// TIA Portal project "Zufallszahl" (V20)

(* hardware
DEVICE "S7-1500/ET200MP-Station_1"  S7-1500 station
   slot 0: "Profilschiene_0"  Rack  6ES7 590-1***0-0AA0
   slot 1: "PLC_1"  CPU 1513-1 PN  6ES7 513-1AM03-0AB0  V4.0
      slot 3: "CPU-Display_1"  6ES7591-1AA00-0AA0
      slot 32768: "PROFINET-Schnittstelle_1"  X1
         slot 32769: "Port_1"  X1 P1
         slot 32770: "Port_2"  X1 P2
      slot 34817: "Virtual CP interface port_1"  Virtual CP interface port  Virtual CP interface port FW V4.0
   slot 2: "DI 16x24VDC BA_1"  DI 16x24VDC BA  6ES7 521-1BH10-0AA0  V1.1
   slot 3: "DQ 16x24VDC/0.5A ST_1"  DQ 16x24VDC/0.5A ST  6ES7 522-1BH00-0AB0  V2.0
   slot 4: "AI 8xU/I/R/RTD BA_2"  AI 8xU/I/R/RTD BA  6ES7 531-7QF00-0AB0  V1.0
   slot 5: "AQ 8xU/I HS_2"  AQ 8xU/I HS  6ES7 532-5HF00-0AB0  V2.2
*)

// ===== PLC "PLC_1"  CPU 1513-1 PN =====

DATA_BLOCK "Zufallszahl_DB"   // DB1
{ S7_Optimized_Access := 'TRUE' }
VERSION : 0.1
// stored: InstanceOfName Zufallszahl
"Zufallszahl"
BEGIN
END_DATA_BLOCK

FUNCTION_BLOCK "Zufallszahl"   // FB1, FBD
{ S7_Optimized_Access := 'TRUE' }
VERSION : 0.1
   VAR
      Zufallszahl_Generator : Struct
         Zufallszahl : DInt;
         Fehler : Struct
            Aktiv : Bool;
            Status : Word;
            UnterfunkionStatus : Word;
         END_STRUCT;
      END_STRUCT;
   END_VAR
   VAR CONSTANT
      Untere_Grenze : DInt := 100;
      Obere_Grenze : DInt := 999;
   END_VAR
BEGIN

REGION Network 1
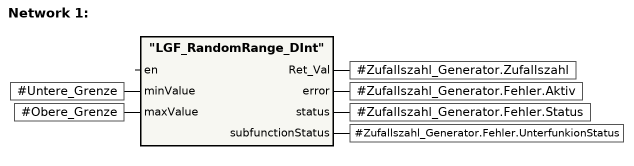
   #Zufallszahl_Generator.Zufallszahl := "LGF_RandomRange_DInt"(minValue := #Untere_Grenze,
                           maxValue := #Obere_Grenze,
                           error => #Zufallszahl_Generator.Fehler.Aktiv,
                           status => #Zufallszahl_Generator.Fehler.Status,
                           subfunctionStatus => #Zufallszahl_Generator.Fehler.UnterfunkionStatus);
END_REGION
END_FUNCTION_BLOCK

ORGANIZATION_BLOCK "Main"   // OB1, FBD, ProgramCycle
TITLE = "Main Program Sweep (Cycle)"
{ S7_Optimized_Access := 'TRUE' }
VERSION : 0.1
   VAR_INPUT
      Initial_Call : Bool;   // Initial call of this OB
      Remanence : Bool;   // =True, if remanent data are available
   END_VAR
   VAR_TEMP
      Aktuelle_Zeit : DTL;
      Fehler : Word;
   END_VAR
BEGIN

REGION Network 1
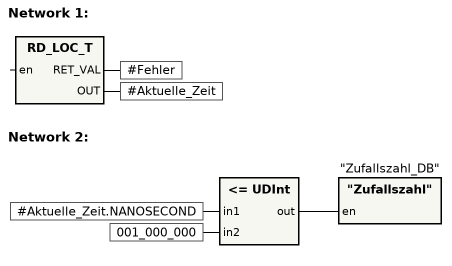
   #Fehler := RD_LOC_T(OUT => #Aktuelle_Zeit);
END_REGION

REGION Network 2
   IF #Aktuelle_Zeit.NANOSECOND <= 001_000_000 THEN
       "Zufallszahl_DB"();   // "Zufallszahl"
   END_IF;
END_REGION
END_ORGANIZATION_BLOCK

// folder: LGF/04 Math operations

FUNCTION "LGF_RandomRange_DInt" : DInt   // FC10013, SCL
TITLE = LGF_RandomRange_DInt
{ S7_Optimized_Access := 'TRUE' }
AUTHOR : Siemens_Digital_Industries
FAMILY : LGF
NAME : LGF_RandomRange_DInt
// This function generates a random value in defined limits with each call.  
// The random number has the data type DInt in the specified range.
// Diese Funktion generiert bei jedem Aufruf einen zufälligen Wert zwischen einem definierten Max- und Minwert.  
// Die Zufallszahl hat den Datentyp DInt im spezifiziertem Wertebereich.
   VAR_INPUT
      minValue : DInt;   // Minimalwert der für den Wertebereich der Zufallszahl - Untergrenze / Minimum value of the range of the random number - lower border
      maxValue : DInt;   // Maximalwert der für den Wertebereich der Zufallszahl - Obergrenze / Maximum value of the range of the random number - upper border
   END_VAR
   VAR_OUTPUT
      error : Bool;   // FALSE: No error TRUE: An error occurred during the execution of the FB / FALSE: Kein Fehler TRUE: Während der Ausführung des FB ist ein Fehler aufgetreten
      status : Word;   // 16#0000-16#7FFF: Status of the FB 16#8000-16#FFFF: Error identification (see following Table) / 16#0000-16#7FFF: Status des FB 16#8000-16#FFFF: Fehleridentifikation (siehe folgende Tabelle)
      subfunctionStatus : Word;   // Status or return value of called FB's, FC's and system blocks / Status oder Rückgabewert von aufgerufenen FB's / FC's und Systemfunktionen
   END_VAR
   VAR_TEMP
      tempTime : DTL;   // Temp memory for System time / Temp variable für System Zeit
      tempNanoSecondInDWord : DWord;   // Temp UDInt converted to DWord for access to individual bytes / Temp UDInt konvertiert nach Dword für den Zufriff per Slice auf die Bytes
      tempTimeStatus : Word;   // Temp status of the instruction `RD_SYS_T` / Temp Status der Systemfunktion `RD_SYS_T`
      tempRandomValue : DWord;   // Temp Random startvalue / Temp Zufallswert als Startwert
      tempNormReal : Real;   // Temp normalized Real value (0.0 - 1.0) / Temp Normalisierer Realwert (0.0 - 1.0)
   END_VAR
   // Ret_Val : Random Real number in the predefined range / Zufallszahl vom Datentyp Real im definierten Wertebereich
   VAR CONSTANT
      ZERO : DInt := 0;   // Zero / 0.0 - value in case of error / Null / 0.0 - Rückgabewert im Fehlerfall
      MAX_UDINT : UDInt := 4294967295 ;   // Maximum DInt datatype / Maximalwert eines DInt Datentype
      SUB_STATUS_NO_ERROR : Word := 16#0000;   // Status: sub function call ends without error / Status: Unterfunktionsaufruf ohne Fehler beendet
      STATUS_FINISHED_NO_ERROR : Word := 16#0000;   // Execution finished without errors / Abarbeitung ohne Fehler beendet
      ERR_MAX_LESS_MIN : Word := 16#8200;   // Error: The ranges specified are wrong: `minValue` is greater than `maxValue` / Fehler: Der spezifizierte Wetebereich is fehlerhaft: `minValue` ist größer als `maxValue`
      ERR_RD_SYS_T : Word := 16#8600;   // Error in `RD_SYS_T` command - check `subFunctionStatus` code / Fehler in Anweisung `RD_SYS_T` - weitere infos in `subFunctionStatus`
   END_VAR
BEGIN
   REGION Block info header
     //=============================================================================
     // SIEMENS AG / (c)Copyright 2017
     //-----------------------------------------------------------------------------
     // Title:            LGF_RandomRange_DInt
     // Comment/Function: This function generates random numbers in defined limits (Datatype DInt)
     // Library/Family:   LGF(Library General Functions)
     // Author:           Siemens Digital Industry Support
     // Tested with:      S7-PLCSIM Advanced V2.0 SP1
     // Engineering:      TIA Portal V15 Update 2
     // Restrictions:     ENO disabled - error handling done by error and status
     // Requirements:     PLC (S7-1200 / S7-1500)
     //-------------------------------------------------------------------------------
     // Change log table:
     // Version  | Date       | Expert in charge       | Changes applied
     //----------|------------|------------------------|------------------------------
     // 01.00.00 19.08.2015  Siemens Industry Online Support
     //                      First released version
     // 01.00.01 02.01.2017  Siemens Industry Online Support
     //                      Upgrade: TIA Portal V14 Update 1
     // 01.00.02 17.08.2018  Siemens Industry Online Support
     //                      Upgrade: TIA V15 Update 2
     // 01.00.03 23.11.2018  Siemens Industry Online Support
     //                      Upgrade: TIA V15.1
     // 01.01.00 09.10.2019  Simatic Systems Support
     //                      Renamed from "LGF_RandomInt" to "LGF_RandomRange_DInt"
     //                      change random datatype from Int to DInt
     //                      Regions, comments and constants are added
     // 03.00.00 23.04.2020  Simatic Systems Support
     //                      Set version to V3.0.0, harmonize the version of the whole library
     // 03.00.01 04.02.2021  Simatic Systems Support
     //                      Insert documentation
     //=============================================================================
   END_REGION Block info header

   REGION DESCRIPTION
     (/*Note
   :    The status of called commands is output in `subFunctionStatus`. In this case, the output value in `status` indicates which command caused the error. In this case, refer to the TIA Portal Online Help section for information on the respective commands.

   The block generates random values that are between the specified `minValue` and the `maxValue`. This random value is output via the `Ret_Val`.

   The random value is formed from the nanoseconds of the current system time of the CPU. The byte order of this value is inverted and then converted to a DInt.
   Hinweis
   :    In `subFunctionStatus` wird der Status von aufgerufenen Anweisungen ausgegeben. Der Ausgangswert in `status` gibt in diesem Fall an, welche Anweisung den Fehler verursacht hat. Holen Sie sich in diesem Fall die Informationen aus der TIA Portal Online Hilfe zu den jeweiligen Anweisungen.

   Der Baustein generiert zufällige Werte, die zwischen dem angegebenen `minValue`-Wert und `maxValue`-Wert liegen. Dieser zufällige Wert wird über den `Ret_Val` ausgegeben.

   Der Zufallswert wird aus den Nanosekunden der aktuellen Systemzeit der CPU gebildet. Dabei wird die Bytereihenfolge dieses Wertes invertiert und anschließend in eine DInt ungewandelt.*/)
   END_REGION DESCRIPTION

   REGION Validation
     // Check if the maximal Value is less than the minimal value
     IF (#minValue > #maxValue) THEN
       #error := true;
       #status := #ERR_MAX_LESS_MIN;
       #subfunctionStatus := #SUB_STATUS_NO_ERROR;
       #LGF_RandomRange_DInt := #ZERO;
       RETURN;
     END_IF;

     // Read system time
     #tempTimeStatus := INT_TO_WORD(RD_SYS_T(#tempTime));

     // Check return variable for error
     IF (#tempTimeStatus <> #SUB_STATUS_NO_ERROR) THEN
       #error := true;
       #status := #ERR_RD_SYS_T;
       #subfunctionStatus := #tempTimeStatus;
       #LGF_RandomRange_DInt := #ZERO;
       RETURN;
     END_IF;
   END_REGION

   REGION Calculating random number
     // Converting to double word so individual bytes can be addressed
     #tempNanoSecondInDWord := UDINT_TO_DWORD(#tempTime.NANOSECOND);

     // Callculate a random-start-value depending on the time
     #tempRandomValue.%B3 := #tempNanoSecondInDWord.%B0;
     #tempRandomValue.%B2 := #tempNanoSecondInDWord.%B1;
     #tempRandomValue.%B1 := #tempNanoSecondInDWord.%B2;
     #tempRandomValue.%B0 := #tempNanoSecondInDWord.%B3;

     // Norm the calculated random number: 0.0 <= #tempNormReal <= 1.0
     #tempNormReal := UDINT_TO_REAL(DWORD_TO_UDINT(#tempRandomValue)) / UDINT_TO_REAL(#MAX_UDINT);

     // Scale the tempNormReal to be in the range of maxValue and minValue
     #LGF_RandomRange_DInt := REAL_TO_DINT((#tempNormReal * DINT_TO_REAL(#maxValue - #minValue) + DINT_TO_REAL(#minValue)));

     #error := false;
     #status := #STATUS_FINISHED_NO_ERROR;
     #subfunctionStatus := #SUB_STATUS_NO_ERROR;
     // ENO mechanism is not used
     ENO := TRUE;
   END_REGION
END_FUNCTION